// TwinCAT 3 PLC project KMWE_Cleanroom_Connect_PLC
// ProgramVersion: 3.1.4024.0
// libraries:
//   KMWE Generic Library, * (KMWE)
//   Tc2_Standard, * (Beckhoff Automation GmbH)
//   Tc2_System, * (Beckhoff Automation GmbH)
//   Tc3_Module, * (Beckhoff Automation GmbH)
// project tree:
//   DUTs/ I_Door.TcIO
//   / PlcTask.TcTTO (not stored)
//   POUs/01 Management layer/HAL/ HAL.TcPOU
//   POUs/04 Control layer/Control %28CM%29/CM_DoorLock/ FB_Flash.TcPOU (not stored), FB_Toggle.TcPOU (not stored), CM_DoorLock.TcPOU (not stored)
//   POUs/04 Control layer/Control %28CM%29/CM_SpeedDoor/ CM_SpeedDoor.TcPOU (not stored), ST_SettingsSpeedDoor.TcDUT (not stored)
//   POUs/04 Control layer/Control %28CM%29/CM_Valve/ CM_Valve.TcPOU (not stored) (excluded from build), ST_ValveFeedback.TcDUT (not stored), ST_ValveFeedback_1.TcDUT (not stored)
//   POUs/ MAIN.TcPOU
// real-time tasks:
//   TASK PlcTask: cycle T#10ms, priority 20, ADS port 350
// I/O:
//   DEVICE Master (EtherCAT) (disabled), AmsNetId 10.130.4.120.2.1
//     Term 1 (EK1200) [EK1200-5000 EtherCAT Power supply (2A E-Bus)]
//       Term 6 (EL6070) [EL6070 1Ch. Licensing-Terminal]
//       Term 2 (EL6900) [EL6900, TwinSAFE PLC]
//       Term 3 (EL1904) [EL1904, 4 Ch. Safety Input 24V, TwinSAFE]
//         modules: Module 1 (FSOES)
//       Term 4 (EL2904) [EL2904, 4 Ch. Safety Output 24V, 0.5A, TwinSAFE]
//         modules: Module 1 (FSOES), Module 2 (DO)
//       Term 7 (EL1008) [EL1008 8Ch. Dig. Input 24V, 3ms]
//       Term 5 (EL9011) [EL9011 End Terminal]
// variable links:
//   Master (EtherCAT) <-> Master (EtherCAT)/Term 1 (EK1200)/Term 2 (EL6900)
//     Term 1 (EK1200)/Term 4 (EL2904)/Module 1 (FSOES)/RxPDO/FSOE <-> ConnectionInputs/TwinSafeGroup1.EL2904, 4 digital outputs_1_4 TxPDO
//     Term 1 (EK1200)/Term 4 (EL2904)/Module 1 (FSOES)/TxPDO/FSOE <-> ConnectionOutputs/TwinSafeGroup1.EL2904, 4 digital outputs_1_4 RxPDO
//   Master (EtherCAT) <-> Master (EtherCAT)/Term 1 (EK1200)/Term 3 (EL1904)
//     Term 1 (EK1200)/Term 2 (EL6900)/ConnectionInputs/TwinSafeGroup1.EL1904, 4 digital inputs_1_3 TxPDO <-> Module 1 (FSOES)/RxPDO/FSOE
//     Term 1 (EK1200)/Term 2 (EL6900)/ConnectionOutputs/TwinSafeGroup1.EL1904, 4 digital inputs_1_3 RxPDO <-> Module 1 (FSOES)/TxPDO/FSOE
//   KMWE_Cleanroom_Connect_PLC/KMWE_Cleanroom_Connect_PLC Instance <-> Master (EtherCAT)/Term 1 (EK1200)/Term 2 (EL6900)
//     PlcTask Outputs/MAIN.Q_SafetyRestart <-> StandardOutputs/TwinSafeGroup1.SafetyRestart_5
//     PlcTask Outputs/MAIN.Q_bErrorAcknowledgement <-> StandardOutputs/TwinSafeGroup1.ErrorAcknowledgement_1
//     PlcTask Outputs/MAIN.Q_bRun <-> StandardOutputs/TwinSafeGroup1.Run_2

// ---- DUTs/I_Door.TcIO
INTERFACE I_Door

METHOD PUBLIC m_Close : BOOL
END_METHOD

METHOD PUBLIC m_Open : BOOL
END_METHOD

METHOD PUBLIC m_Reset : BOOL
END_METHOD

METHOD PUBLIC m_Stop : BOOL
END_METHOD

{attribute 'monitoring':='call'}
PROPERTY PUBLIC p_bStaIsClosed : BOOL
GET
END_GET
END_PROPERTY

{attribute 'monitoring':='call'}
PROPERTY PUBLIC p_bStaIsClosing : BOOL
GET
END_GET
END_PROPERTY

{attribute 'monitoring':='call'}
PROPERTY PUBLIC p_bStaIsOpened : BOOL
GET
END_GET
END_PROPERTY

{attribute 'monitoring':='call'}
PROPERTY PUBLIC p_bStaIsOpening : BOOL
GET
END_GET
END_PROPERTY

END_INTERFACE

// ---- POUs/01 Management layer/HAL/HAL.TcPOU
FUNCTION_BLOCK HAL


//--{attribute 'TcLinkTo' := 'TIID^Master (EtherCAT)^Term 1 (EK1200)^Term 7 (EL1008)^Channel 1^Input'}
//--     bVarIn2    AT%I*  : BOOL;  // linked via attribute

END_FUNCTION_BLOCK

// ---- POUs/MAIN.TcPOU
PROGRAM MAIN
VAR

	// Control Module SIM/TEST
	cmSpeedDoorOuter : CM_SpeedDoor;
	arr_bTestBoolSpeeddoor : ARRAY[0..15] OF BOOL;
	arr_bTestCmdSpeeddoor : ARRAY[0..15] OF BOOL;
	
	CmDoorLockCleanroomDoor : CM_DoorLock;
	arr_bTestBoolCleanroomDoor : ARRAY[0..15] OF BOOL;
	arr_bTestCmdCleanroomDoor : ARRAY[0..15] OF BOOL;
	
	cmValveDoorUnlockingPinUpper : CM_Valve;
	cmValveDoorUnlockingPinLower : CM_Valve;
	
	cmValveDockingClampsUpper : CM_Valve;
	cmValveDockingClampsLower : CM_Valve;
	arr_bTestBoolValve : ARRAY[0..15] OF BOOL;
	arr_bTestCmdValve : ARRAY[0..15] OF BOOL;

	// PLC --> SAFETY IO
	Q_bErrorAcknowledgement AT %Q* : BOOL;
	Q_bRun AT %Q* : BOOL;
	Q_SafetyRestart AT %Q* : BOOL;
END_VAR

// Speed Door simulation/test
cmSpeedDoorOuter(
	i_bReqEnable := arr_bTestCmdSpeeddoor[10],
	i_eCtrlMode := E_CtrlMode.AUTOMATIC,
	i_bCmdReset := arr_bTestCmdSpeeddoor[11],
	i_sCmName := 'Speeddoor Outer');

IF arr_bTestCmdSpeeddoor[0] THEN cmSpeedDoorOuter.m_Open(); arr_bTestCmdSpeeddoor[0] := FALSE; END_IF;
IF arr_bTestCmdSpeeddoor[1] THEN cmSpeedDoorOuter.m_Close(); arr_bTestCmdSpeeddoor[1] := FALSE; END_IF;
IF arr_bTestCmdSpeeddoor[2] THEN cmSpeedDoorOuter.m_Reset(); arr_bTestCmdSpeeddoor[2] := FALSE; END_IF;
IF arr_bTestCmdSpeeddoor[3] THEN cmSpeedDoorOuter.m_Stop(); arr_bTestCmdSpeeddoor[3] := FALSE; END_IF;

arr_bTestBoolSpeeddoor[0] := cmSpeedDoorOuter.p_bStaEnabled;
arr_bTestBoolSpeeddoor[1] := cmSpeedDoorOuter.p_bStaError;
arr_bTestBoolSpeeddoor[2] := cmSpeedDoorOuter.p_bStaIsOpening;
arr_bTestBoolSpeeddoor[3] := cmSpeedDoorOuter.p_bStaIsOpened;
arr_bTestBoolSpeeddoor[4] := cmSpeedDoorOuter.p_bStaIsClosing;
arr_bTestBoolSpeeddoor[5] := cmSpeedDoorOuter.p_bStaIsClosed;

// Cleanroom Door simulation/test
CmDoorLockCleanroomDoor(
	i_bReqEnable := arr_bTestCmdCleanroomDoor[10],
	i_eCtrlMode := E_CtrlMode.AUTOMATIC,
	i_bCmdReset := arr_bTestCmdCleanroomDoor[11],
	i_sCmName := 'Speeddoor Outer');

IF arr_bTestCmdCleanroomDoor[0] THEN cmDoorLockCleanroomDoor.m_Release(); arr_bTestCmdCleanroomDoor[0] := FALSE; END_IF;
IF arr_bTestCmdCleanroomDoor[1] THEN cmDoorlockCleanroomDoor.m_Apply(); arr_bTestCmdCleanroomDoor[1] := FALSE; END_IF;

arr_bTestBoolCleanroomDoor[0] := cmDoorLockCleanroomDoor.p_bStaEnabled;
arr_bTestBoolCleanroomDoor[1] := cmDoorLockCleanroomDoor.p_bStaError;
arr_bTestBoolCleanroomDoor[2] := cmDoorLockCleanroomDoor.p_bReqReleaseLock;
arr_bTestBoolCleanroomDoor[3] := cmDoorLockCleanroomDoor.p_bStaDoorIsClosed;
arr_bTestBoolCleanroomDoor[4] := cmDoorLockCleanroomDoor.p_bStaLockIsApplied;
arr_bTestBoolCleanroomDoor[5] := cmDoorLockCleanroomDoor.p_bStaLockIsReleased;

// Valves simulation/test
cmValveDockingClampsUpper(
	i_bReqEnable := arr_bTestCmdValve[10],
	i_eCtrlMode := E_CtrlMode.AUTOMATIC,
	i_bCmdReset := arr_bTestCmdValve[11],
	i_sCmName := 'Docking Clamp Upper');
	
cmValveDockingClampsLower(
	i_bReqEnable := arr_bTestCmdValve[12],
	i_eCtrlMode := E_CtrlMode.AUTOMATIC,
	i_bCmdReset := arr_bTestCmdValve[13],
	i_sCmName := 'Docking Clamp Lower');

END_PROGRAM
